{region '#Template'}
	{attribute 'Version' := '5.0.0.0'}
	{attribute 'Tags' := '"LCID": "1031", "Text": "Universal, Analog, Aggregate"'}
	{attribute 'Tags' := '"LCID": "1033", "Text": "Universal, Analog, Aggregate"'}
	{attribute 'Using' := '"Type": "Template", "URI": "EC_ID"'}
	{attribute 'Using' := '"Type": "Template", "URI": "BA2_Param"'}
	{attribute 'Description' := '"LCID": "1031", "Text": "AV"'}
	{attribute 'Description' := '"LCID": "1033", "Text": "AV"'}
{endregion}
FUNCTION_BLOCK FB_BA_ActuatorAV EXTENDS FB_BA_View
VAR_INPUT
	stCmd					: ST_BA_Analog;	
END_VAR
VAR_OUTPUT
	fPresentValue		: REAL;
	bDst				: BOOL;
	eActivePrio			: E_BA_Priority;	
END_VAR
VAR_INPUT CONSTANT
	Val					: FB_BA_AV;		
	PlantLock			: FB_BA_PlantLock;	
END_VAR
VAR
	bPrioSfty				: BOOL;
	bPrioCrit				: BOOL;	
END_VAR

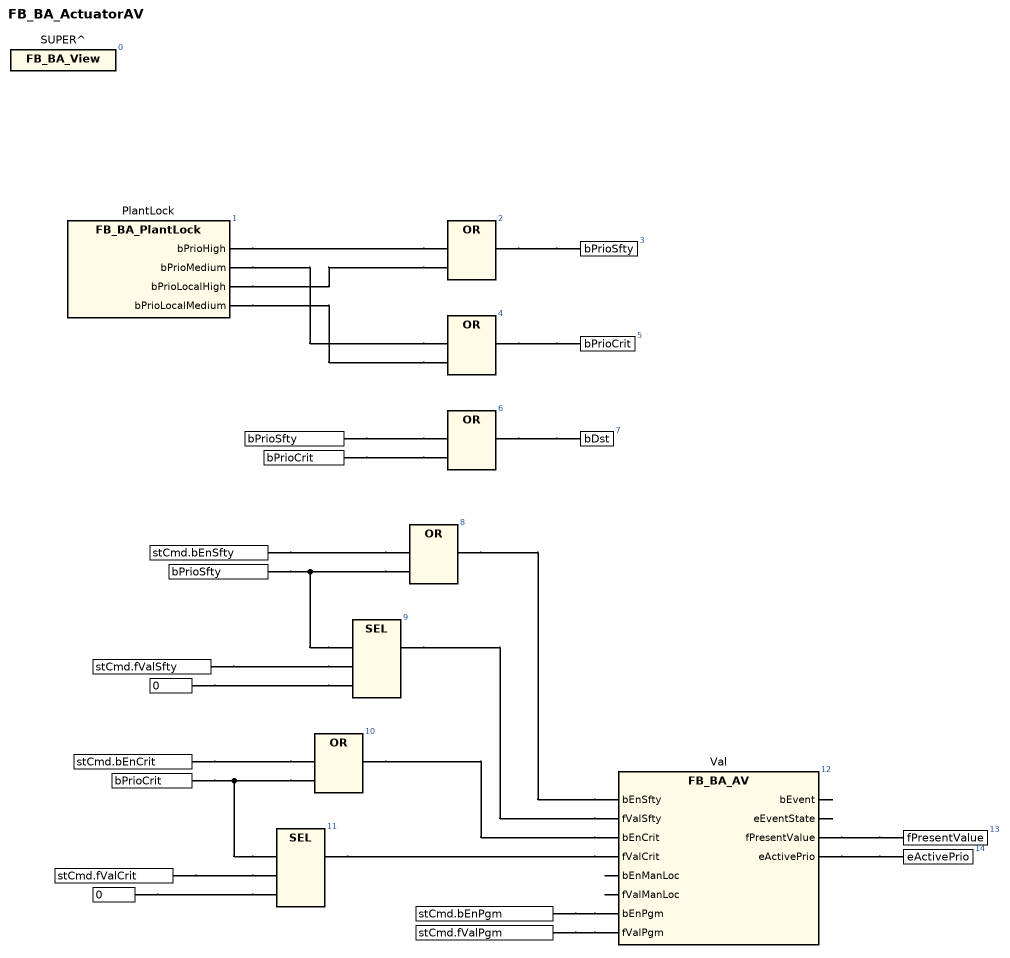
SUPER^(); // FB_BA_View
PlantLock(); // FB_BA_PlantLock
bPrioSfty := PlantLock.bPrioHigh OR PlantLock.bPrioLocalHigh;
bPrioCrit := PlantLock.bPrioMedium OR PlantLock.bPrioLocalMedium;
bDst := bPrioSfty OR bPrioCrit;
Val(
    bEnSfty := stCmd.bEnSfty OR bPrioSfty,
    fValSfty := SEL(bPrioSfty, stCmd.fValSfty, 0),
    bEnCrit := stCmd.bEnCrit OR bPrioCrit,
    fValCrit := SEL(bPrioCrit, stCmd.fValCrit, 0),
    bEnPgm := stCmd.bEnPgm,
    fValPgm := stCmd.fValPgm); // FB_BA_AV
fPresentValue := Val.fPresentValue;
eActivePrio := Val.eActivePrio;

METHOD FB_init : BOOL
VAR_INPUT
	bInitRetains : BOOL; // if TRUE, the retain variables are initialized (warm start / cold start)
	bInCopyCode : BOOL;  // if TRUE, the instance afterwards gets moved into the copy code (online change)
END_VAR
PlantLock.Parent				:= THIS^;		

Val.iParent						:= THIS^;
Val.iLabel						:= LblFun_ControlSignal;  
Val.eUnit						:= E_BA_Unit.eOther_Percent;
Val.fCOVIncrement				:= BA2_Param.fDefCOVIncrement;
Val.bEnManualRm					:= FALSE;	//	Priority  8	
Val.fValManualRm				:= 0.0;		//	Priority  8
Val.fDefaultValue				:= 0.0;	
Val.nEventClassID				:= EC_ID.NC80;
Val.stTimeDelay.nToNormal		:= BA2_Param.nDefTimeDelay_ToNormal;
Val.stTimeDelay.nToAbnormal		:= BA2_Param.nDefTimeDelay_ToAbnormal;
Val.stHighLimit.bEnable			:= FALSE;
Val.stHighLimit.fValue			:= 0.0;		
Val.stLowLimit.bEnable			:= FALSE;
Val.stLowLimit.fValue			:= 0.0;
Val.fLimitDeadband 				:= BA2_Param.fDefLimitDeadband;
Val.bAcknowledgeRm				:= FALSE;	
Val.aEventTransitionText[1]		:= txtEvent_Disturb;
Val.aEventTransitionText[2]		:= txtEvent_None;
Val.aEventTransitionText[3]		:= txtEvent_Normal;
Val.bEventDetectionEnable		:= FALSE;
Val.eEnPlantLock				:= E_BA_LockPriority.eNoLock;
END_METHOD

END_FUNCTION_BLOCK

(* stored: Version 1.1.0.1, ProductVersion 3.1.4024.12
   POU FB_BA_ActuatorAV: Id {a6413a34-102e-43f8-b665-3b065a31562e}, SpecialFunc None
   Method FB_init: Id {ee128fe4-5d4f-42a2-8fba-e436e9cc8744} *)
